// TwinCAT 3 PLC project Tests
// ProgramVersion: 3.1.4023.0
// libraries:
//   Tc2_Standard, * (Beckhoff Automation GmbH)
//   Tc2_System, * (Beckhoff Automation GmbH)
//   Tc3_Module, * (Beckhoff Automation GmbH)
//   TcUnit, * (www.tcunit.org)
// project tree:
//   FBs to test/FBs/ FB_Co2FlowModelDeviationHandler.TcPOU, FB_ConsumptionCalculator.TcPOU, FB_mF.TcPOU, FB_MovingAverage.TcPOU, FB_StateSpaceModel.TcPOU
//   FBs to test/ITFs/ I_TON.TcIO
//   FBs to test/Wrappers/ TON_Wrapper.TcPOU
//   / PlcTask.TcTTO
//   Unit Tests/FB tests/ FB_Co2FlowModelDeviationHandler_Test.TcPOU, FB_ConsumptionCalculator_Test.TcPOU, FB_mF_Test.TcPOU, FB_MovingAverage_Test.TcPOU
//   Unit Tests/Mocks/ TON_Mock_TimerRanOut.TcPOU (not stored)
//   Unit Tests/ TESTS_MAIN.TcPOU
// (motion and I/O tree: see PLC project untitled1)
// real-time tasks:
//   TASK PlcTask: cycle T#10ms, priority 20, ADS port 350
//   TASK VISU_TASK: cycle T#200000us, priority 30, ADS port 351
//   TASK PlcTaskFast: cycle T#2ms, priority 1, ADS port 352
//   TASK PlcTask1: cycle T#10ms, priority 21, ADS port 353
// variable links:

CONFIGURATION Tests
    RESOURCE PLC ON TwinCAT3
        TASK PlcTask(INTERVAL := T#10ms, PRIORITY := 21);
        PROGRAM TESTS_MAIN WITH PlcTask : TESTS_MAIN;
    END_RESOURCE
END_CONFIGURATION

// ---- FBs to test/ITFs/I_TON.TcIO
INTERFACE I_TON

METHOD Call : BOOL
VAR_INPUT
    IN 	: BOOL;
    PT 	: TIME;
END_VAR
VAR_OUTPUT
	Q 	: BOOL;
	ET 	: TIME;
END_VAR
END_METHOD

END_INTERFACE

// ---- Unit Tests/TESTS_MAIN.TcPOU
 PROGRAM TESTS_MAIN
VAR
	startTests : BOOL;
	
	// FBs to test
	fbMovingAverageTest : FB_MovingAverage_Test;
	fbConsumptionCalculatorTest : FB_ConsumptionCalculator_Test;
	fbmFTest : FB_mF_Test;
	fbCo2ModelDeviationHandlerTest : FB_Co2FlowModelDeviationHandler_Test;
	movingavg : FB_MovingAverage;
	consumptioncalc : FB_ConsumptionCalculator;
	measF : REAL;
	
	mF : FB_mF;
	TON_Test : TON;
	meas : LREAL;
	uTest : ARRAY[1..15] OF LREAL;
	fbGetCurTaskIndex : GETCURTASKINDEX;
END_VAR


fbGetCurTaskIndex();
IF _TaskInfo[fbGetCurTaskIndex.index].FirstCycle THEN
    // The code that you want to be executed at the first cycle
	mF.Init(
		activateObserver := FALSE);
END_IF

IF startTests THEN
	TcUnit.RUN();
	movingavg.startCalculation(
							start := TRUE,
							measurement := meas,
							intervalS := 1,
							windowS := 10,
							dTime := T#10MS,
							excludeUntilReady := FALSE);
	consumptioncalc.calculate(
							start := TRUE,
							valuePerSec := movingavg.value/60,
							intervalS := 10,
							dtime := T#10MS);
	uTest[1];
	TON_Test(IN := TRUE, PT := T#1S);
	IF TON_Test.Q THEN
		mF.Step(
				u := uTest,
				y_meas := meas);
		TON_Test(IN := FALSE);
		mF.y[1];
	END_IF
END_IF

END_PROGRAM

// ---- Unit Tests/FB tests/FB_MovingAverage_Test.TcPOU
FUNCTION_BLOCK FB_MovingAverage_Test EXTENDS TcUnit.FB_TestSuite

calculationShouldBeReadyWhenTimePassed();
calculationShouldNotBeReadyBeforeTimePassed();
movingAverageOfThreePlusTwoPlusOneShouldBeTwo();
resetMethodCallShouldResetValue();
theValueShouldBe40AfterTwoSeconds();
valueShouldBe0BeforeWindowPassedIfPreReadyNotIncluded();

METHOD calculationShouldBeReadyWhenTimePassed : BOOL
VAR
	movingAverage : FB_MovingAverage;
END_VAR

TEST('calculationShouldBeReadyWhenTimePassed');
movingAverage.startCalculation(TRUE,0, 3,1, T#3S, FALSE);
AssertEquals_BOOL(Expected := TRUE, Actual :=  movingAverage.ready, Message := 'Moving average calculation not ready after time passed');
TEST_FINISHED();
END_METHOD

METHOD calculationShouldNotBeReadyBeforeTimePassed : BOOL
VAR
	movingAverage : FB_MovingAverage;
END_VAR

TEST('calculationShouldNotBeReadyBeforeTimePassed');
movingAverage.startCalculation(TRUE, 0, 1,1, T#0S, FALSE);
AssertEquals_BOOL(Expected := FALSE, Actual :=  movingAverage.ready, Message := 'Moving average calculation ready before time passed');
TEST_FINISHED();
END_METHOD

METHOD movingAverageOfThreePlusTwoPlusOneShouldBeTwo
VAR
	movingAverage : FB_MovingAverage;
END_VAR

TEST('movingAverageOfThreePlusTwoPlusOneShouldBeTwo');
movingAverage.startCalculation(TRUE, 3, 3, 1, T#1S, FALSE);
movingAverage.startCalculation(TRUE, 2, 3, 1, T#1S, FALSE);
movingAverage.startCalculation(TRUE, 1, 3, 1, T#1S, FALSE);
movingAverage.startCalculation(TRUE, 0, 3, 1, T#1S, FALSE);
AssertEquals_REAL(Expected := 2, Actual := movingAverage.value, 0, Message := 'Moving average calculation not equal to two!');
TEST_FINISHED();
END_METHOD

METHOD resetMethodCallShouldResetValue
VAR
	movingAverage : FB_MovingAverage;
END_VAR

TEST('resetMethodCallShouldResetValue');
movingAverage.startCalculation(start := TRUE, measurement := 50, intervalS := 1, windowS := 3, dtime := T#3S, excludeUntilReady := FALSE);
movingAverage.reset();
AssertEquals_REAL(0, movingAverage.value, 0, 'Reset did not reset value!'); 
TEST_FINISHED();
END_METHOD

METHOD theValueShouldBe40AfterTwoSeconds
VAR
	movingAverage : FB_MovingAverage;
END_VAR
TEST('theValueShouldBe40AfterTwoSeconds');
movingAverage.startCalculation(start := TRUE, measurement := 40, intervalS := 1, windowS := 3, dtime := T#1S, excludeUntilReady := FALSE);
movingAverage.startCalculation(start := TRUE, measurement := 40, intervalS := 1, windowS := 3, dtime := T#1S, excludeUntilReady := FALSE);
AssertEquals_REAL(40, movingAverage.value, 0, 'Value not 40 after two seconds'); 
TEST_FINISHED();
END_METHOD

METHOD valueShouldBe0BeforeWindowPassedIfPreReadyNotIncluded
VAR
	movingAverage : FB_MovingAverage;
END_VAR

TEST('valueShouldBe0BeforeWindowPassedIfPreReadyNotIncluded');
movingAverage.startCalculation(start := TRUE, measurement := 40, intervalS := 1, windowS := 3, dtime := T#1S, excludeUntilReady := TRUE);
movingAverage.startCalculation(start := TRUE, measurement := 40, intervalS := 1, windowS := 3, dtime := T#1S, excludeUntilReady := TRUE);
AssertEquals_REAL(0, movingAverage.value, 0, 'Value not 0 before window passed when exclude values before first window checked'); 
TEST_FINISHED();
END_METHOD

END_FUNCTION_BLOCK

// ---- FBs to test/FBs/FB_MovingAverage.TcPOU
FUNCTION_BLOCK FB_MovingAverage
VAR_OUTPUT
	ready : BOOL;
	value : REAL;
END_VAR
VAR
    sum           : REAL;
    count         : UDINT;
    running       : BOOL;
    elapsedTime   : TIME;
	
	addToSum		: BOOL;
	elapsedSecond	: INT;
	valueArray		: ARRAY[1..999] OF REAL;
	i				: INT;
	
    intervalTime : TIME;
END_VAR

METHOD reset : BOOL
VAR_INPUT
END_VAR

value := 0;
ready := FALSE;
sum := 0;
count := 0;
running := FALSE;
elapsedTime := T#0S;
elapsedSecond := 0;
FOR i := 1 TO 999 DO
	valueArray[i] := 0;
END_FOR
END_METHOD

METHOD startCalculation : BOOL
VAR_INPUT
    start : BOOL;
    measurement : REAL;
    windowS : INT;
	intervalS : INT;
    dtime : TIME;  
	excludeUntilReady : BOOL;
END_VAR

// If window is 0, return immediately
IF windowS = 0 THEN
	RETURN;
END_IF

// Start edge
IF start AND NOT running THEN
    running := TRUE;
END_IF

IF running THEN
	elapsedTime := elapsedTime + dtime;
	intervalTime := intervalTime + dtime;
	
	// Every second, calculate new mean value and shift values forward
	IF ready THEN
		IF (TIME_TO_INT(intervalTime))/1000 >= intervalS THEN
			addToSum := TRUE;
			elapsedSecond := elapsedSecond + 1;
			FOR i := 1 TO windowS DO
				sum := sum + valueArray[i];
			END_FOR
			value := sum/windowS;
			// Shift values
			FOR i := 1 TO windowS - 1 DO
				valueArray[i] := valueArray[i + 1];
			END_FOR
			valueArray[windowS] := measurement;
			intervalTime := T#0S;
			sum := 0;
		END_IF
	ELSE
		IF (TIME_TO_INT(intervalTime))/1000 >= intervalS THEN
			elapsedSecond := elapsedSecond + 1;
			valueArray[elapsedSecond] := measurement;
			intervalTime := T#0S;
			IF NOT excludeUntilReady THEN
				FOR i := 1 TO elapsedSecond DO
					sum := sum + valueArray[i];
				END_FOR
				value := sum / elapsedSecond;
				sum := 0;
			ELSE
				value := 0;
			END_IF
		END_IF
	END_IF
	
	// After initial interval passed, start calculating the value
	IF elapsedTime >= INT_TO_TIME(windowS*1000) THEN
		startCalculation := TRUE;
		ready := TRUE;
	END_IF
	
END_IF
END_METHOD

END_FUNCTION_BLOCK

// ---- Unit Tests/FB tests/FB_ConsumptionCalculator_Test.TcPOU
FUNCTION_BLOCK FB_ConsumptionCalculator_Test EXTENDS TcUnit.FB_TestSuite
VAR_INPUT
END_VAR
VAR_OUTPUT
END_VAR
VAR
END_VAR

theCalculatedValueShouldBeTenAfterTenSeconds();
theCalculatedValueShouldBe20After20Seconds();
theCalulatedValueShouldBe30After20Seconds();

METHOD theCalculatedValueShouldBe20After20Seconds
VAR
	consumptionCalc : FB_ConsumptionCalculator;
END_VAR

TEST('theCalculatedValueShouldBe20After20Seconds');

consumptionCalc.calculate(
						start := TRUE,
						valuePerSec := 1,
						intervalS := 10,
						dtime := T#10S);
consumptionCalc.sum;								
consumptionCalc.calculate(
						start := TRUE,
						valuePerSec := 1,
						intervalS := 10,
						dtime := T#10S);
consumptionCalc.sum;			
						
AssertEquals_REAL(Expected := 20, Actual := consumptionCalc.sum, Delta := 0, Message := 'Calculated value not twenty after twenty seconds');

consumptionCalc.reset();
AssertEquals_REAL(Expected := 0, Actual := consumptionCalc.sum, Delta := 0, Message := 'Calculated value not reset');

TEST_FINISHED();
END_METHOD

METHOD theCalculatedValueShouldBeTenAfterTenSeconds : BOOL
VAR
	consumptionCalc : FB_ConsumptionCalculator;
END_VAR

TEST('theCalculatedValueShouldBeTenAfterTenSeconds');
consumptionCalc.calculate(
						start := TRUE,
						valuePerSec := 0,
						intervalS := 10,
						dtime := T#10MS);
	
consumptionCalc.sum;						
consumptionCalc.calculate(
						start := TRUE,
						valuePerSec := 1,
						intervalS := 10,
						dtime := T#10S);
consumptionCalc.sum;
						
AssertEquals_REAL(Expected := 10, Actual := consumptionCalc.sum, Delta := 0, Message := 'Calculated value not ten after ten seconds');

TEST_FINISHED();
END_METHOD

METHOD theCalulatedValueShouldBe30After20Seconds
VAR
	consumptionCalc : FB_ConsumptionCalculator;
END_VAR

TEST('theCalulatedValueShouldBe30After20Seconds');

consumptionCalc.calculate(
						start := TRUE,
						valuePerSec := 1,
						intervalS := 10,
						dtime := T#10S);
						
consumptionCalc.calculate(
						start := TRUE,
						valuePerSec := 2,
						intervalS := 10,
						dtime := T#10S);

AssertEquals_REAL(Expected := 30, Actual := consumptionCalc.sum, Delta := 0, Message := 'Calculated value not 30 after twenty seconds');


TEST_FINISHED();
END_METHOD

END_FUNCTION_BLOCK

// ---- FBs to test/FBs/FB_ConsumptionCalculator.TcPOU
FUNCTION_BLOCK FB_ConsumptionCalculator
VAR_INPUT
END_VAR
VAR_OUTPUT
	sum : REAL;
END_VAR
VAR
    running       : BOOL;
    elapsedTime   : TIME;
	RTRIG_Started : R_TRIG;
	amountOfCycles: DINT;
	counter : DINT;
END_VAR

METHOD calculate : BOOL
VAR_INPUT
	start : BOOL;
	valuePerSec : REAL;
    intervalS : INT;
    dtime : TIME;   
END_VAR
VAR
    intervalTime : TIME;
END_VAR
intervalTime := INT_TO_TIME(intervalS*1000);
RTRIG_Started(CLK := start);
// Start edge
IF RTRIG_Started.q THEN
    running := TRUE;
    sum := 0.0;
    elapsedTime := T#0S;
END_IF

IF NOT start THEN
	running := FALSE;
END_IF

IF running THEN
	// Simulate time passing
	elapsedTime := elapsedTime + dtime;
	IF elapsedTime >= intervalTime THEN
		sum := sum + valuePerSec*(intervalS);
		elapsedTime := T#0S;
		amountOfCycles := amountOfCycles + counter;
		counter := 0;
	END_IF 
	counter := counter + 1;
END_IF
END_METHOD

METHOD reset : BOOL
VAR_INPUT
END_VAR

sum := 0;
running := FALSE;
elapsedTime := T#0S;
counter := 0;
amountOfCycles := 0;
END_METHOD

END_FUNCTION_BLOCK

// ---- Unit Tests/FB tests/FB_mF_Test.TcPOU
FUNCTION_BLOCK FB_mF_Test EXTENDS TcUnit.FB_TestSuite


valueShouldChangeWhenInputChanges();

METHOD valueShouldChangeWhenInputChanges
VAR
	mF : FB_mF;
	uTest : ARRAY[1..15] OF LREAL;
END_VAR

TEST('valueShouldChangeWhenInputChanges');
	uTest[1] := 5;
	mF.Step(
			u := uTest,
			y_meas := 2);
TEST_FINISHED();
END_METHOD

END_FUNCTION_BLOCK

// ---- FBs to test/FBs/FB_mF.TcPOU
FUNCTION_BLOCK FB_mF EXTENDS FB_StateSpaceModel
VAR_INPUT
END_VAR
VAR_OUTPUT
END_VAR
VAR
END_VAR

METHOD PUBLIC Init
VAR_INPUT
	activateObserver : BOOL;
END_VAR
VAR
    i,j : INT;
END_VAR

SUPER^();
nx := 2;
nu := 2;
ny := 1;

// Load matrices
_A[1,1] := 0.9895;
_A[1,2] := 0.03677;
_A[2,1] := -0.01237;
_A[2,2] := 0.9649;

_B[1,1] := -2.52E-05;
_B[1,2] := -1.673E-06;
_B[2,1] := -2.199E-04;
_B[2,2] := -5.346E-06;

_C[1,1] := -10.22;
_C[1,2] := -0.1235;

_K[1] := -0.1242;
_K[2] := -0.5091;
END_METHOD

END_FUNCTION_BLOCK

// ---- FBs to test/FBs/FB_StateSpaceModel.TcPOU
FUNCTION_BLOCK ABSTRACT FB_StateSpaceModel
VAR
    nx : INT;
    nu : INT;
    ny : INT;
	
    x  		: ARRAY[1..15] OF LREAL;

    _A  : ARRAY[1..15,1..15] OF LREAL;
    _B  : ARRAY[1..15,1..15] OF LREAL;
    _C  : ARRAY[1..15,1..15] OF LREAL;
    _D  : ARRAY[1..15,1..15] OF LREAL;
    _K  : ARRAY[1..15] OF LREAL;

	_activateObserver : BOOL;
    bInit : BOOL;
	
	i,j : INT;
    x_new : ARRAY[1..10] OF LREAL;
    e : LREAL;
END_VAR
VAR_OUTPUT
	y  : ARRAY[1..15] OF LREAL;
END_VAR

METHOD PUBLIC Init
VAR_INPUT
	activateObserver : BOOL;
END_VAR
VAR
    i,j : INT;
END_VAR

FOR i := 1 TO nx DO
    x[i] := 0;
    _K[i] := _K[i]; // keep
END_FOR
_activateObserver := activateObserver;
bInit := TRUE;
END_METHOD

METHOD PUBLIC Step
VAR_INPUT
    u  		: ARRAY[1..15] OF LREAL;
	y_meas 	: LREAL;
END_VAR

// --- Output ---
FOR i := 1 TO ny DO
    y[i] := 0;
    FOR j := 1 TO nx DO 
        y[i] := y[i] + _C[i,j]*x[j];
    END_FOR
END_FOR

// --- Innovation (single y example) ---
IF _activateObserver THEN
	e := y_meas - y[1];
ELSE 
	e := 0;
END_IF

// --- State update ---
FOR i := 1 TO nx DO
    x_new[i] := 0;

    FOR j := 1 TO nx DO
        x_new[i] := x_new[i] + _A[i,j]*x[j];
    END_FOR

    FOR j := 1 TO nu DO
        x_new[i] := x_new[i] + _B[i,j]*u[j];
    END_FOR

    x_new[i] := x_new[i] + _K[i]*e;
END_FOR

FOR i := 1 TO nx DO
    x[i] := x_new[i];
END_FOR
END_METHOD

END_FUNCTION_BLOCK

// ---- Unit Tests/FB tests/FB_Co2FlowModelDeviationHandler_Test.TcPOU
FUNCTION_BLOCK FB_Co2FlowModelDeviationHandler_Test EXTENDS TcUnit.FB_TestSuite
VAR_INPUT
END_VAR
VAR_OUTPUT
END_VAR
VAR
END_VAR


simpleCalculationsTest();
ifCurrentFlowIsZeroDeviationShouldBeZero();

METHOD ifCurrentFlowIsZeroDeviationShouldBeZero
VAR
	deviationHandler : FB_Co2FlowModelDeviationHandler;
END_VAR

TEST('ifCurrentFlowIsZeroDeviationShouldBeZero');

deviationHandler(
			currentFlow := 0,
			modeledFlow := 50);
					
AssertEquals_DINT(Expected := 0, Actual := deviationHandler.deviationPercentage, Message := 'Deviation not zero when current flow is zero');

TEST_FINISHED();
END_METHOD

METHOD simpleCalculationsTest
VAR
	deviationHandler : FB_Co2FlowModelDeviationHandler;
END_VAR

TEST('deviationShouldBeMinus50');

deviationHandler(
			currentFlow := 100,
			modeledFlow := 50);
					
AssertEquals_DINT(Expected := -50, Actual := deviationHandler.deviationPercentage, Message := 'Deviation not -50 when it should be');

TEST_FINISHED();

TEST('deviationShouldBePlus20');

deviationHandler(
			currentFlow := 100,
			modeledFlow := 120);
					
AssertEquals_DINT(Expected := 20, Actual := deviationHandler.deviationPercentage, Message := 'Deviation not 20 when it should be');

TEST_FINISHED();
END_METHOD

END_FUNCTION_BLOCK

// ---- FBs to test/FBs/FB_Co2FlowModelDeviationHandler.TcPOU
FUNCTION_BLOCK FB_Co2FlowModelDeviationHandler
VAR_INPUT
	currentFlow : REAL;
	modeledFlow : REAL;
END_VAR
VAR_OUTPUT
	deviationPercentage : DINT;
END_VAR
VAR
	delta : REAL;
END_VAR


IF currentFlow <> 0 THEN
	delta := modeledFlow / currentFlow;
	
	IF delta < 0 THEN
		deviationPercentage := TO_DINT(delta*100);
	ELSE
		deviationPercentage := TO_DINT(-(100 - delta*100));
	END_IF
	
ELSE
	currentFlow := 0;
END_IF

END_FUNCTION_BLOCK

// ---- FBs to test/Wrappers/TON_Wrapper.TcPOU
FUNCTION_BLOCK TON_Wrapper implements I_TON
VAR
    {attribute 'hide'} _ton : TON;
    {attribute 'hide'} _q 	: BOOL;
   	{attribute 'hide'} _et 	: TIME;
END_VAR

 
METHOD Call : BOOL
VAR_INPUT
	IN	: BOOL;
	PT	: TIME;
END_VAR
VAR_OUTPUT
	Q 	: BOOL;
	ET 	: TIME;
END_VAR

_ton(IN := IN, PT := PT);
Q := _ton.Q;
ET := _ton.ET;
END_METHOD

END_FUNCTION_BLOCK
